{attribute 'TcGenerated'}
{attribute 'no-analysis'}
{attribute 'linkalways'}
// This function has been automatically generated from the project information.
VAR_GLOBAL CONSTANT
	{attribute 'const_non_replaced'}
	stLibVersion_Tc3_BAR_Common : ST_LibVersion := (iMajor := 0, iMinor := 4, iBuild := 0, iRevision := 0, nFlags := 0, sVersion := '0.2.1');
END_VAR

(* stored: Version 1.1.0.1, ProductVersion 3.1.4024.9
   GVL Global_Version: Id {629dd8fe-5783-484b-af5a-b41584f4330c} *)
